// TIA Portal V19 export
FUNCTION "A04_TrkManager_CALL" : Void   // FC98, LAD
// stored: SetENOAutomatically false
BEGIN

REGION Network 1
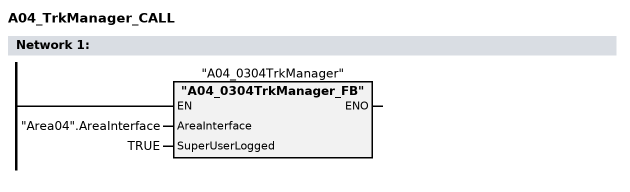
   RUNG wire#powerrail
      "A04_0304TrkManager"(AreaInterface := "Area04".AreaInterface, SuperUserLogged := TRUE)
   END_RUNG
   // the same network as SCL:
   "A04_0304TrkManager"(AreaInterface := "Area04".AreaInterface, SuperUserLogged := TRUE);   // "A04_0304TrkManager_FB"
END_REGION
END_FUNCTION
